// TIA Portal V18 export
TYPE "DO"
// stored: IsFailsafeCompliant false
   STRUCT
      BUZZER : Bool;
      "BFV 1" : Bool;
      "BFV 2" : Bool;
      "BFV 3" : Bool;
      "BFV 4" : Bool;
      "BFV 5" : Bool;
      "BFV 6" : Bool;
      "BFV 7" : Bool;
      "BFV 8" : Bool;
      "BFV 9" : Bool;
      R1 : Bool;
      R2 : Bool;
      R3 : Bool;
      R4 : Bool;
      R5 : Bool;
      R6 : Bool;
      "BFV 10" : Bool;
      "BFV 11" : Bool;
      "BFV 12" : Bool;
      "BFV 13" : Bool;
      "BFV 14" : Bool;
      "BFV 15" : Bool;
      "BFV 16" : Bool;
      "BFV 17" : Bool;
      "BFV 18" : Bool;
      "BFV 19" : Bool;
      "CIP SUPPLY PUMP START (VFD)" : Bool;
      "ACID DOSING PUMP" : Bool;
      "CAUSTIC DOSING PUMP" : Bool;
      "RETURN PUMP 1" : Bool;
      "RETURN PUMP 2" : Bool;
      "RETUEN PUMP 3" : Bool;
   END_STRUCT;
END_TYPE
